PROGRAM MAIN
VAR
END_VAR

END_PROGRAM

(* stored: Version 1.1.0.1
   POU MAIN: Id {4038daf6-7c5e-4628-9780-6d75915f1fc2} *)
